// TIA Portal V19 export
// export: Created 2026-04-27T21:44:43.6095817Z, ExportSetting None, DisplayName Totally Integrated Automation Portal, DisplayVersion V19, DisplayName TIA Portal Openness, DisplayVersion V19, DisplayName TIA Portal Version Control Interface, DisplayVersion V19, DisplayName STEP 7 Professional, DisplayVersion V19, DisplayName STEP 7 Safety, DisplayVersion V19, DisplayName WinCC Basic/Comfort/Advanced, DisplayVersion V19, DisplayName WinCC Unified, DisplayVersion V19
FUNCTION "Process_Temp" : Void   // FC1, LAD
{ S7_Optimized_Access := 'TRUE' }
// stored: SetENOAutomatically false
BEGIN

REGION Network 2: TI-10112-TI
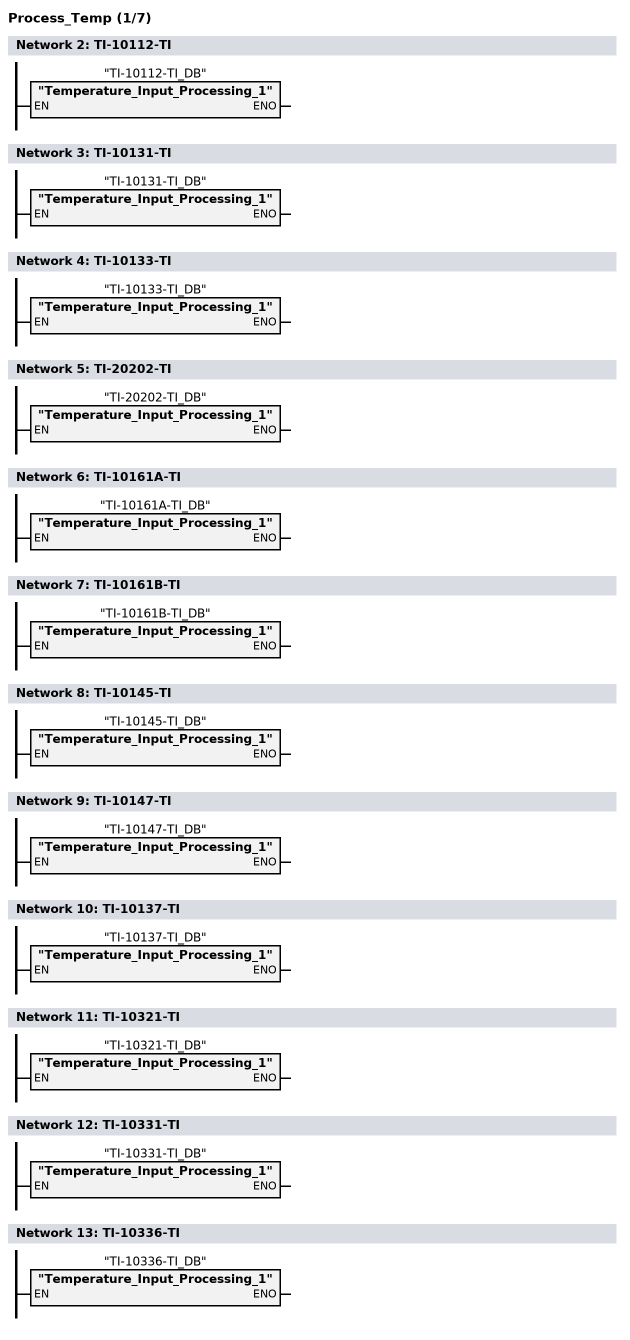
   RUNG wire#powerrail
      "TI-10112-TI_DB"()
   END_RUNG
   // the same network as SCL:
   "TI-10112-TI_DB"();   // "Temperature_Input_Processing_1"
END_REGION

REGION Network 3: TI-10131-TI
   RUNG wire#powerrail
      "TI-10131-TI_DB"()
   END_RUNG
   // the same network as SCL:
   "TI-10131-TI_DB"();   // "Temperature_Input_Processing_1"
END_REGION

REGION Network 4: TI-10133-TI
   RUNG wire#powerrail
      "TI-10133-TI_DB"()
   END_RUNG
   // the same network as SCL:
   "TI-10133-TI_DB"();   // "Temperature_Input_Processing_1"
END_REGION

REGION Network 5: TI-20202-TI
   RUNG wire#powerrail
      "TI-20202-TI_DB"()
   END_RUNG
   // the same network as SCL:
   "TI-20202-TI_DB"();   // "Temperature_Input_Processing_1"
END_REGION

REGION Network 6: TI-10161A-TI
   RUNG wire#powerrail
      "TI-10161A-TI_DB"()
   END_RUNG
   // the same network as SCL:
   "TI-10161A-TI_DB"();   // "Temperature_Input_Processing_1"
END_REGION

REGION Network 7: TI-10161B-TI
   RUNG wire#powerrail
      "TI-10161B-TI_DB"()
   END_RUNG
   // the same network as SCL:
   "TI-10161B-TI_DB"();   // "Temperature_Input_Processing_1"
END_REGION

REGION Network 8: TI-10145-TI
   RUNG wire#powerrail
      "TI-10145-TI_DB"()
   END_RUNG
   // the same network as SCL:
   "TI-10145-TI_DB"();   // "Temperature_Input_Processing_1"
END_REGION

REGION Network 9: TI-10147-TI
   RUNG wire#powerrail
      "TI-10147-TI_DB"()
   END_RUNG
   // the same network as SCL:
   "TI-10147-TI_DB"();   // "Temperature_Input_Processing_1"
END_REGION

REGION Network 10: TI-10137-TI
   RUNG wire#powerrail
      "TI-10137-TI_DB"()
   END_RUNG
   // the same network as SCL:
   "TI-10137-TI_DB"();   // "Temperature_Input_Processing_1"
END_REGION

REGION Network 11: TI-10321-TI
   RUNG wire#powerrail
      "TI-10321-TI_DB"()
   END_RUNG
   // the same network as SCL:
   "TI-10321-TI_DB"();   // "Temperature_Input_Processing_1"
END_REGION

REGION Network 12: TI-10331-TI
   RUNG wire#powerrail
      "TI-10331-TI_DB"()
   END_RUNG
   // the same network as SCL:
   "TI-10331-TI_DB"();   // "Temperature_Input_Processing_1"
END_REGION

REGION Network 13: TI-10336-TI
   RUNG wire#powerrail
      "TI-10336-TI_DB"()
   END_RUNG
   // the same network as SCL:
   "TI-10336-TI_DB"();   // "Temperature_Input_Processing_1"
END_REGION

REGION Network 14: TI-20113-TI
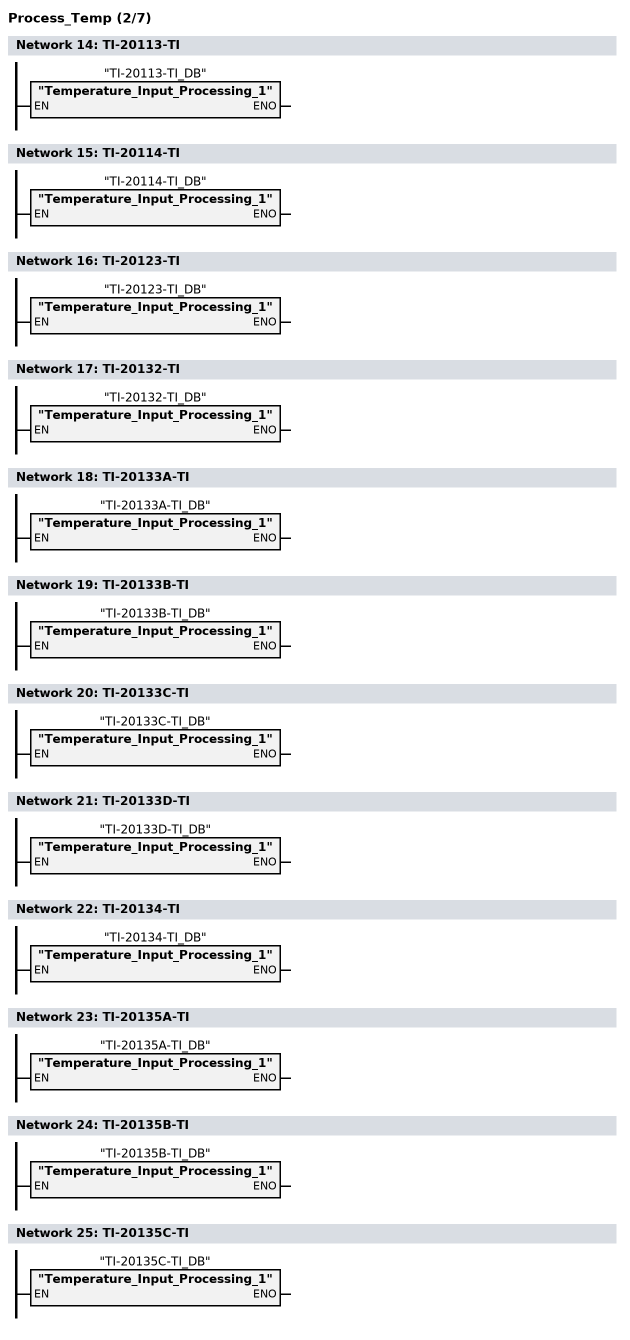
   RUNG wire#powerrail
      "TI-20113-TI_DB"()
   END_RUNG
   // the same network as SCL:
   "TI-20113-TI_DB"();   // "Temperature_Input_Processing_1"
END_REGION

REGION Network 15: TI-20114-TI
   RUNG wire#powerrail
      "TI-20114-TI_DB"()
   END_RUNG
   // the same network as SCL:
   "TI-20114-TI_DB"();   // "Temperature_Input_Processing_1"
END_REGION

REGION Network 16: TI-20123-TI
   RUNG wire#powerrail
      "TI-20123-TI_DB"()
   END_RUNG
   // the same network as SCL:
   "TI-20123-TI_DB"();   // "Temperature_Input_Processing_1"
END_REGION

REGION Network 17: TI-20132-TI
   RUNG wire#powerrail
      "TI-20132-TI_DB"()
   END_RUNG
   // the same network as SCL:
   "TI-20132-TI_DB"();   // "Temperature_Input_Processing_1"
END_REGION

REGION Network 18: TI-20133A-TI
   RUNG wire#powerrail
      "TI-20133A-TI_DB"()
   END_RUNG
   // the same network as SCL:
   "TI-20133A-TI_DB"();   // "Temperature_Input_Processing_1"
END_REGION

REGION Network 19: TI-20133B-TI
   RUNG wire#powerrail
      "TI-20133B-TI_DB"()
   END_RUNG
   // the same network as SCL:
   "TI-20133B-TI_DB"();   // "Temperature_Input_Processing_1"
END_REGION

REGION Network 20: TI-20133C-TI
   RUNG wire#powerrail
      "TI-20133C-TI_DB"()
   END_RUNG
   // the same network as SCL:
   "TI-20133C-TI_DB"();   // "Temperature_Input_Processing_1"
END_REGION

REGION Network 21: TI-20133D-TI
   RUNG wire#powerrail
      "TI-20133D-TI_DB"()
   END_RUNG
   // the same network as SCL:
   "TI-20133D-TI_DB"();   // "Temperature_Input_Processing_1"
END_REGION

REGION Network 22: TI-20134-TI
   RUNG wire#powerrail
      "TI-20134-TI_DB"()
   END_RUNG
   // the same network as SCL:
   "TI-20134-TI_DB"();   // "Temperature_Input_Processing_1"
END_REGION

REGION Network 23: TI-20135A-TI
   RUNG wire#powerrail
      "TI-20135A-TI_DB"()
   END_RUNG
   // the same network as SCL:
   "TI-20135A-TI_DB"();   // "Temperature_Input_Processing_1"
END_REGION

REGION Network 24: TI-20135B-TI
   RUNG wire#powerrail
      "TI-20135B-TI_DB"()
   END_RUNG
   // the same network as SCL:
   "TI-20135B-TI_DB"();   // "Temperature_Input_Processing_1"
END_REGION

REGION Network 25: TI-20135C-TI
   RUNG wire#powerrail
      "TI-20135C-TI_DB"()
   END_RUNG
   // the same network as SCL:
   "TI-20135C-TI_DB"();   // "Temperature_Input_Processing_1"
END_REGION

REGION Network 26: TI-20135D-TI
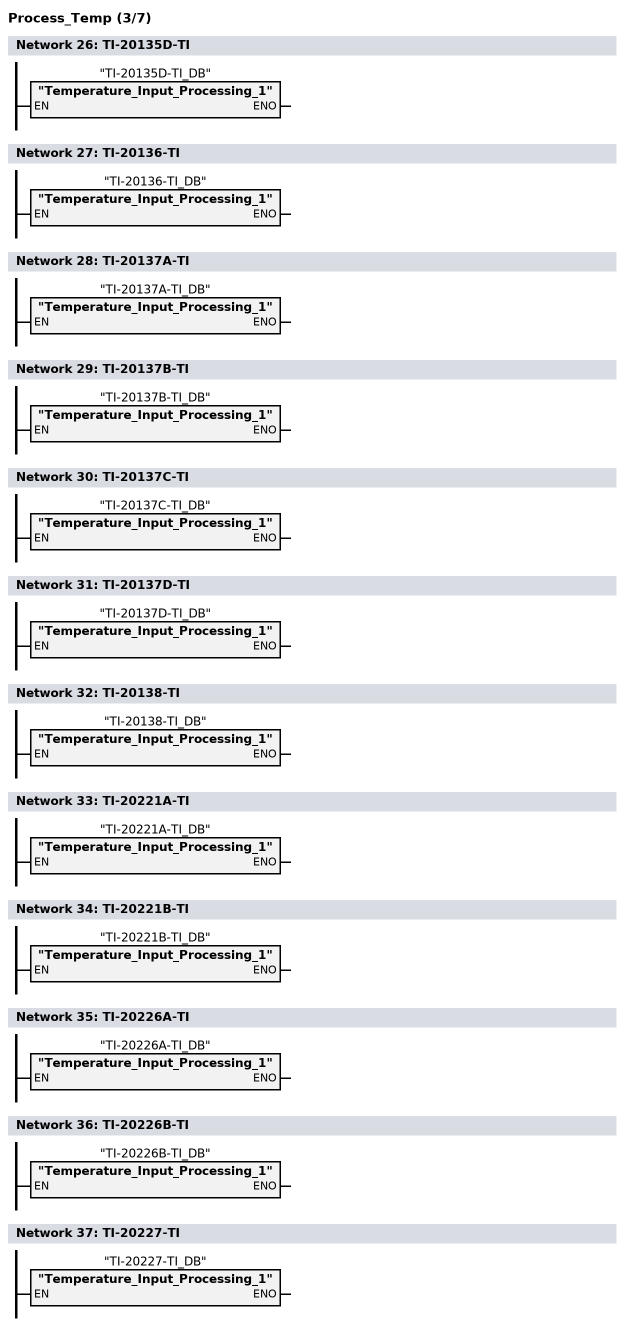
   RUNG wire#powerrail
      "TI-20135D-TI_DB"()
   END_RUNG
   // the same network as SCL:
   "TI-20135D-TI_DB"();   // "Temperature_Input_Processing_1"
END_REGION

REGION Network 27: TI-20136-TI
   RUNG wire#powerrail
      "TI-20136-TI_DB"()
   END_RUNG
   // the same network as SCL:
   "TI-20136-TI_DB"();   // "Temperature_Input_Processing_1"
END_REGION

REGION Network 28: TI-20137A-TI
   RUNG wire#powerrail
      "TI-20137A-TI_DB"()
   END_RUNG
   // the same network as SCL:
   "TI-20137A-TI_DB"();   // "Temperature_Input_Processing_1"
END_REGION

REGION Network 29: TI-20137B-TI
   RUNG wire#powerrail
      "TI-20137B-TI_DB"()
   END_RUNG
   // the same network as SCL:
   "TI-20137B-TI_DB"();   // "Temperature_Input_Processing_1"
END_REGION

REGION Network 30: TI-20137C-TI
   RUNG wire#powerrail
      "TI-20137C-TI_DB"()
   END_RUNG
   // the same network as SCL:
   "TI-20137C-TI_DB"();   // "Temperature_Input_Processing_1"
END_REGION

REGION Network 31: TI-20137D-TI
   RUNG wire#powerrail
      "TI-20137D-TI_DB"()
   END_RUNG
   // the same network as SCL:
   "TI-20137D-TI_DB"();   // "Temperature_Input_Processing_1"
END_REGION

REGION Network 32: TI-20138-TI
   RUNG wire#powerrail
      "TI-20138-TI_DB"()
   END_RUNG
   // the same network as SCL:
   "TI-20138-TI_DB"();   // "Temperature_Input_Processing_1"
END_REGION

REGION Network 33: TI-20221A-TI
   RUNG wire#powerrail
      "TI-20221A-TI_DB"()
   END_RUNG
   // the same network as SCL:
   "TI-20221A-TI_DB"();   // "Temperature_Input_Processing_1"
END_REGION

REGION Network 34: TI-20221B-TI
   RUNG wire#powerrail
      "TI-20221B-TI_DB"()
   END_RUNG
   // the same network as SCL:
   "TI-20221B-TI_DB"();   // "Temperature_Input_Processing_1"
END_REGION

REGION Network 35: TI-20226A-TI
   RUNG wire#powerrail
      "TI-20226A-TI_DB"()
   END_RUNG
   // the same network as SCL:
   "TI-20226A-TI_DB"();   // "Temperature_Input_Processing_1"
END_REGION

REGION Network 36: TI-20226B-TI
   RUNG wire#powerrail
      "TI-20226B-TI_DB"()
   END_RUNG
   // the same network as SCL:
   "TI-20226B-TI_DB"();   // "Temperature_Input_Processing_1"
END_REGION

REGION Network 37: TI-20227-TI
   RUNG wire#powerrail
      "TI-20227-TI_DB"()
   END_RUNG
   // the same network as SCL:
   "TI-20227-TI_DB"();   // "Temperature_Input_Processing_1"
END_REGION

REGION Network 38: TI-20228-TI
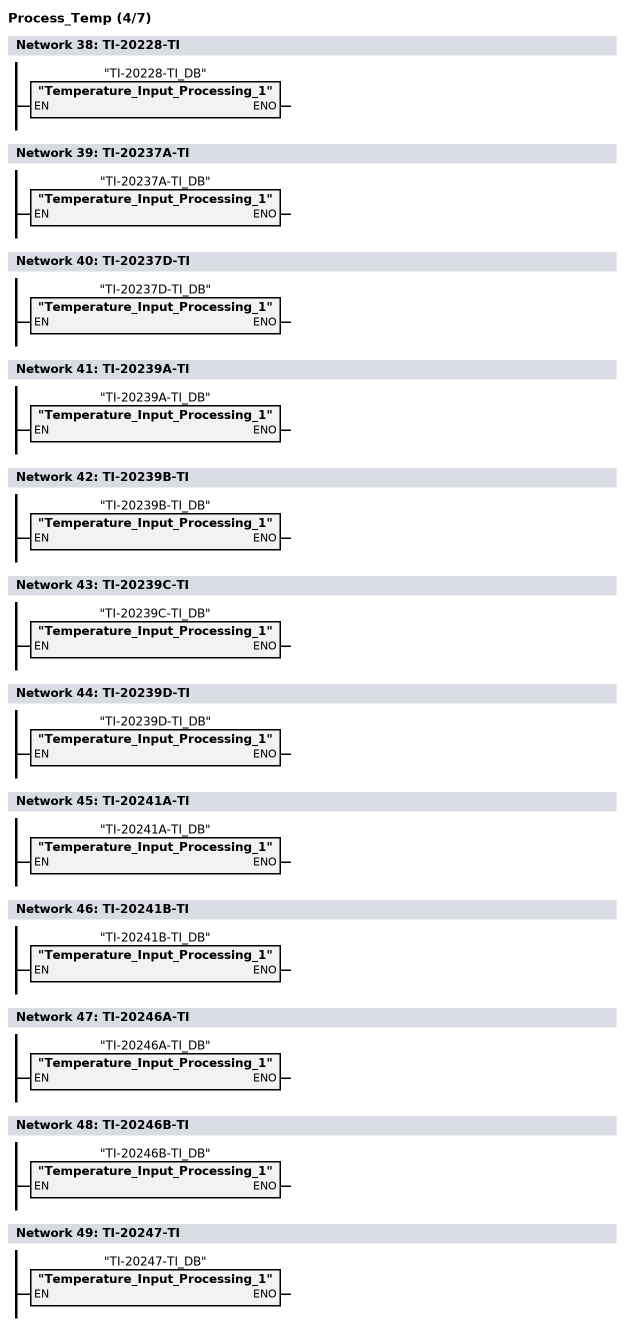
   RUNG wire#powerrail
      "TI-20228-TI_DB"()
   END_RUNG
   // the same network as SCL:
   "TI-20228-TI_DB"();   // "Temperature_Input_Processing_1"
END_REGION

REGION Network 39: TI-20237A-TI
   RUNG wire#powerrail
      "TI-20237A-TI_DB"()
   END_RUNG
   // the same network as SCL:
   "TI-20237A-TI_DB"();   // "Temperature_Input_Processing_1"
END_REGION

REGION Network 40: TI-20237D-TI
   RUNG wire#powerrail
      "TI-20237D-TI_DB"()
   END_RUNG
   // the same network as SCL:
   "TI-20237D-TI_DB"();   // "Temperature_Input_Processing_1"
END_REGION

REGION Network 41: TI-20239A-TI
   RUNG wire#powerrail
      "TI-20239A-TI_DB"()
   END_RUNG
   // the same network as SCL:
   "TI-20239A-TI_DB"();   // "Temperature_Input_Processing_1"
END_REGION

REGION Network 42: TI-20239B-TI
   RUNG wire#powerrail
      "TI-20239B-TI_DB"()
   END_RUNG
   // the same network as SCL:
   "TI-20239B-TI_DB"();   // "Temperature_Input_Processing_1"
END_REGION

REGION Network 43: TI-20239C-TI
   RUNG wire#powerrail
      "TI-20239C-TI_DB"()
   END_RUNG
   // the same network as SCL:
   "TI-20239C-TI_DB"();   // "Temperature_Input_Processing_1"
END_REGION

REGION Network 44: TI-20239D-TI
   RUNG wire#powerrail
      "TI-20239D-TI_DB"()
   END_RUNG
   // the same network as SCL:
   "TI-20239D-TI_DB"();   // "Temperature_Input_Processing_1"
END_REGION

REGION Network 45: TI-20241A-TI
   RUNG wire#powerrail
      "TI-20241A-TI_DB"()
   END_RUNG
   // the same network as SCL:
   "TI-20241A-TI_DB"();   // "Temperature_Input_Processing_1"
END_REGION

REGION Network 46: TI-20241B-TI
   RUNG wire#powerrail
      "TI-20241B-TI_DB"()
   END_RUNG
   // the same network as SCL:
   "TI-20241B-TI_DB"();   // "Temperature_Input_Processing_1"
END_REGION

REGION Network 47: TI-20246A-TI
   RUNG wire#powerrail
      "TI-20246A-TI_DB"()
   END_RUNG
   // the same network as SCL:
   "TI-20246A-TI_DB"();   // "Temperature_Input_Processing_1"
END_REGION

REGION Network 48: TI-20246B-TI
   RUNG wire#powerrail
      "TI-20246B-TI_DB"()
   END_RUNG
   // the same network as SCL:
   "TI-20246B-TI_DB"();   // "Temperature_Input_Processing_1"
END_REGION

REGION Network 49: TI-20247-TI
   RUNG wire#powerrail
      "TI-20247-TI_DB"()
   END_RUNG
   // the same network as SCL:
   "TI-20247-TI_DB"();   // "Temperature_Input_Processing_1"
END_REGION

REGION Network 50: TI-20248-TI
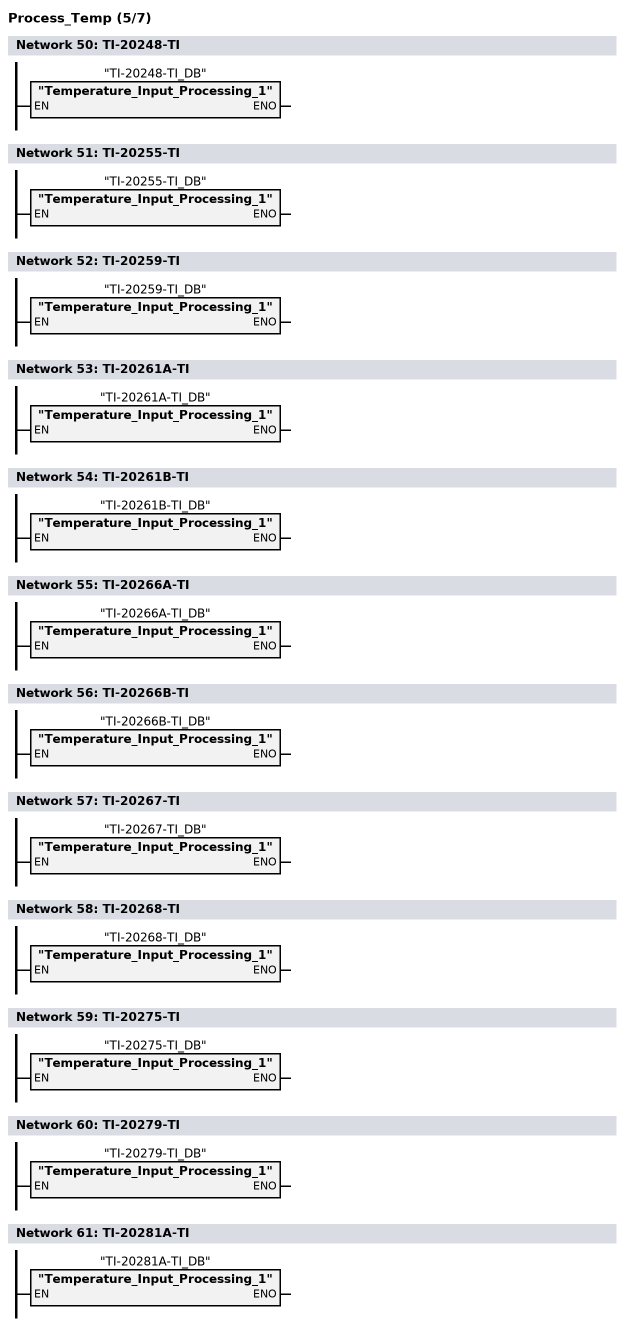
   RUNG wire#powerrail
      "TI-20248-TI_DB"()
   END_RUNG
   // the same network as SCL:
   "TI-20248-TI_DB"();   // "Temperature_Input_Processing_1"
END_REGION

REGION Network 51: TI-20255-TI
   RUNG wire#powerrail
      "TI-20255-TI_DB"()
   END_RUNG
   // the same network as SCL:
   "TI-20255-TI_DB"();   // "Temperature_Input_Processing_1"
END_REGION

REGION Network 52: TI-20259-TI
   RUNG wire#powerrail
      "TI-20259-TI_DB"()
   END_RUNG
   // the same network as SCL:
   "TI-20259-TI_DB"();   // "Temperature_Input_Processing_1"
END_REGION

REGION Network 53: TI-20261A-TI
   RUNG wire#powerrail
      "TI-20261A-TI_DB"()
   END_RUNG
   // the same network as SCL:
   "TI-20261A-TI_DB"();   // "Temperature_Input_Processing_1"
END_REGION

REGION Network 54: TI-20261B-TI
   RUNG wire#powerrail
      "TI-20261B-TI_DB"()
   END_RUNG
   // the same network as SCL:
   "TI-20261B-TI_DB"();   // "Temperature_Input_Processing_1"
END_REGION

REGION Network 55: TI-20266A-TI
   RUNG wire#powerrail
      "TI-20266A-TI_DB"()
   END_RUNG
   // the same network as SCL:
   "TI-20266A-TI_DB"();   // "Temperature_Input_Processing_1"
END_REGION

REGION Network 56: TI-20266B-TI
   RUNG wire#powerrail
      "TI-20266B-TI_DB"()
   END_RUNG
   // the same network as SCL:
   "TI-20266B-TI_DB"();   // "Temperature_Input_Processing_1"
END_REGION

REGION Network 57: TI-20267-TI
   RUNG wire#powerrail
      "TI-20267-TI_DB"()
   END_RUNG
   // the same network as SCL:
   "TI-20267-TI_DB"();   // "Temperature_Input_Processing_1"
END_REGION

REGION Network 58: TI-20268-TI
   RUNG wire#powerrail
      "TI-20268-TI_DB"()
   END_RUNG
   // the same network as SCL:
   "TI-20268-TI_DB"();   // "Temperature_Input_Processing_1"
END_REGION

REGION Network 59: TI-20275-TI
   RUNG wire#powerrail
      "TI-20275-TI_DB"()
   END_RUNG
   // the same network as SCL:
   "TI-20275-TI_DB"();   // "Temperature_Input_Processing_1"
END_REGION

REGION Network 60: TI-20279-TI
   RUNG wire#powerrail
      "TI-20279-TI_DB"()
   END_RUNG
   // the same network as SCL:
   "TI-20279-TI_DB"();   // "Temperature_Input_Processing_1"
END_REGION

REGION Network 61: TI-20281A-TI
   RUNG wire#powerrail
      "TI-20281A-TI_DB"()
   END_RUNG
   // the same network as SCL:
   "TI-20281A-TI_DB"();   // "Temperature_Input_Processing_1"
END_REGION

REGION Network 62: TI-20281B-TI
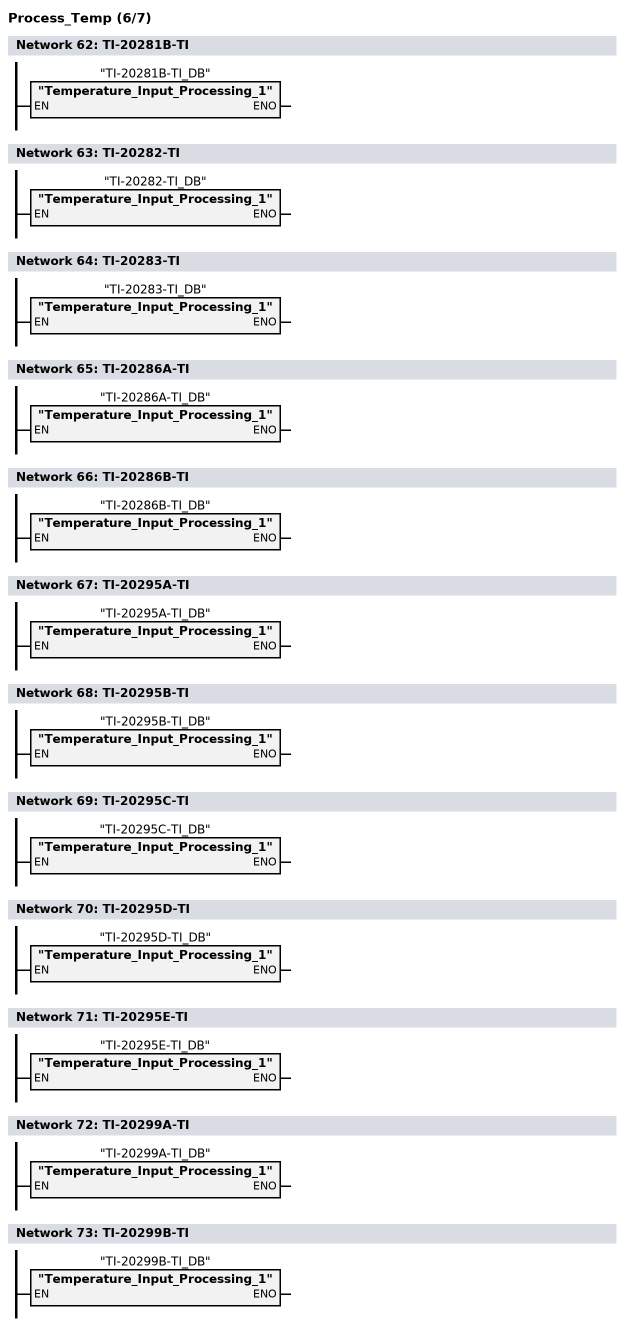
   RUNG wire#powerrail
      "TI-20281B-TI_DB"()
   END_RUNG
   // the same network as SCL:
   "TI-20281B-TI_DB"();   // "Temperature_Input_Processing_1"
END_REGION

REGION Network 63: TI-20282-TI
   RUNG wire#powerrail
      "TI-20282-TI_DB"()
   END_RUNG
   // the same network as SCL:
   "TI-20282-TI_DB"();   // "Temperature_Input_Processing_1"
END_REGION

REGION Network 64: TI-20283-TI
   RUNG wire#powerrail
      "TI-20283-TI_DB"()
   END_RUNG
   // the same network as SCL:
   "TI-20283-TI_DB"();   // "Temperature_Input_Processing_1"
END_REGION

REGION Network 65: TI-20286A-TI
   RUNG wire#powerrail
      "TI-20286A-TI_DB"()
   END_RUNG
   // the same network as SCL:
   "TI-20286A-TI_DB"();   // "Temperature_Input_Processing_1"
END_REGION

REGION Network 66: TI-20286B-TI
   RUNG wire#powerrail
      "TI-20286B-TI_DB"()
   END_RUNG
   // the same network as SCL:
   "TI-20286B-TI_DB"();   // "Temperature_Input_Processing_1"
END_REGION

REGION Network 67: TI-20295A-TI
   RUNG wire#powerrail
      "TI-20295A-TI_DB"()
   END_RUNG
   // the same network as SCL:
   "TI-20295A-TI_DB"();   // "Temperature_Input_Processing_1"
END_REGION

REGION Network 68: TI-20295B-TI
   RUNG wire#powerrail
      "TI-20295B-TI_DB"()
   END_RUNG
   // the same network as SCL:
   "TI-20295B-TI_DB"();   // "Temperature_Input_Processing_1"
END_REGION

REGION Network 69: TI-20295C-TI
   RUNG wire#powerrail
      "TI-20295C-TI_DB"()
   END_RUNG
   // the same network as SCL:
   "TI-20295C-TI_DB"();   // "Temperature_Input_Processing_1"
END_REGION

REGION Network 70: TI-20295D-TI
   RUNG wire#powerrail
      "TI-20295D-TI_DB"()
   END_RUNG
   // the same network as SCL:
   "TI-20295D-TI_DB"();   // "Temperature_Input_Processing_1"
END_REGION

REGION Network 71: TI-20295E-TI
   RUNG wire#powerrail
      "TI-20295E-TI_DB"()
   END_RUNG
   // the same network as SCL:
   "TI-20295E-TI_DB"();   // "Temperature_Input_Processing_1"
END_REGION

REGION Network 72: TI-20299A-TI
   RUNG wire#powerrail
      "TI-20299A-TI_DB"()
   END_RUNG
   // the same network as SCL:
   "TI-20299A-TI_DB"();   // "Temperature_Input_Processing_1"
END_REGION

REGION Network 73: TI-20299B-TI
   RUNG wire#powerrail
      "TI-20299B-TI_DB"()
   END_RUNG
   // the same network as SCL:
   "TI-20299B-TI_DB"();   // "Temperature_Input_Processing_1"
END_REGION

REGION Network 74: TI-20299C-TI
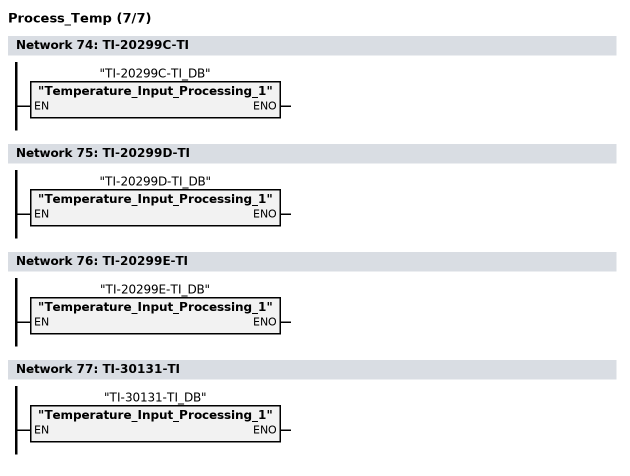
   RUNG wire#powerrail
      "TI-20299C-TI_DB"()
   END_RUNG
   // the same network as SCL:
   "TI-20299C-TI_DB"();   // "Temperature_Input_Processing_1"
END_REGION

REGION Network 75: TI-20299D-TI
   RUNG wire#powerrail
      "TI-20299D-TI_DB"()
   END_RUNG
   // the same network as SCL:
   "TI-20299D-TI_DB"();   // "Temperature_Input_Processing_1"
END_REGION

REGION Network 76: TI-20299E-TI
   RUNG wire#powerrail
      "TI-20299E-TI_DB"()
   END_RUNG
   // the same network as SCL:
   "TI-20299E-TI_DB"();   // "Temperature_Input_Processing_1"
END_REGION

REGION Network 77: TI-30131-TI
   RUNG wire#powerrail
      "TI-30131-TI_DB"()
   END_RUNG
   // the same network as SCL:
   "TI-30131-TI_DB"();   // "Temperature_Input_Processing_1"
END_REGION
END_FUNCTION
